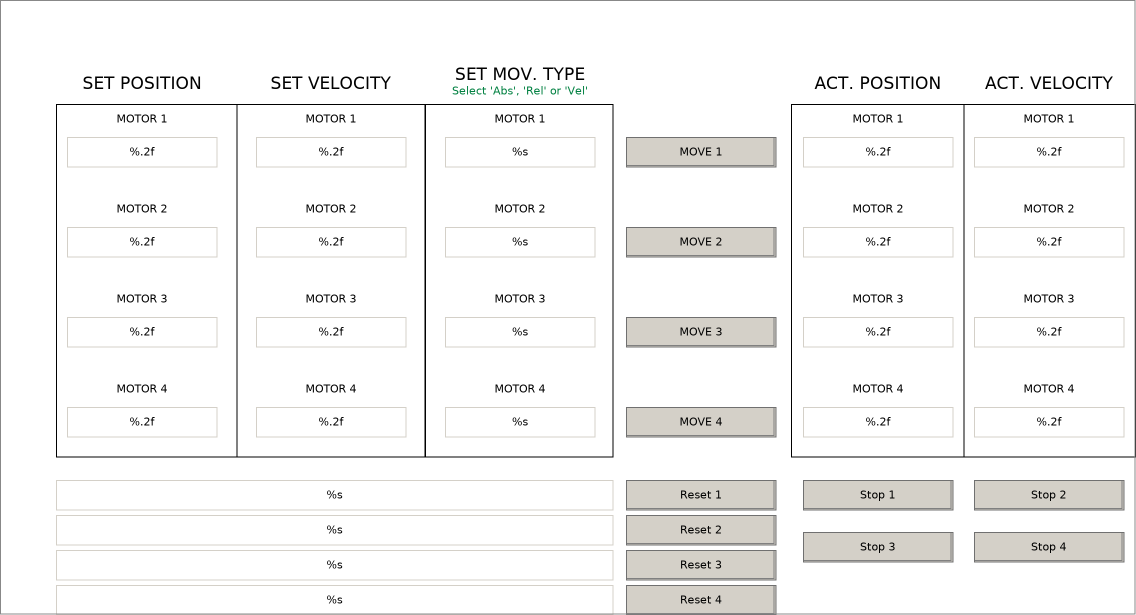
VISUALIZATION Visualization  // 1136x615
    Rectangle (425,104 188x353)
    Rectangle (233,104 192x353)
    Rectangle (56,104 181x353)
    Textfield (67,137 150x30), "%.2f", text variable: MAIN.lrPosition[1]
        OnMouseClick: write the text variable via Default
    Label (67,104 150x30), "MOTOR 1"
    Textfield (67,227 150x30), "%.2f", text variable: MAIN.lrPosition[2]
        OnMouseClick: write the text variable via Default
    Label (67,194 150x30), "MOTOR 2"
    Textfield (67,317 150x30), "%.2f", text variable: MAIN.lrPosition[3]
        OnMouseClick: write the text variable via Default
    Label (67,284 150x30), "MOTOR 3"
    Textfield (67,407 150x30), "%.2f", text variable: MAIN.lrPosition[4]
        OnMouseClick: write the text variable via Default
    Label (67,374 150x30), "MOTOR 4"
    Textfield (256,137 150x30), "%.2f", text variable: MAIN.lrVelocity[1]
        OnMouseClick: write the text variable via Default
    Label (256,104 150x30), "MOTOR 1"
    Textfield (256,227 150x30), "%.2f", text variable: MAIN.lrVelocity[2]
        OnMouseClick: write the text variable via Default
    Label (256,194 150x30), "MOTOR 2"
    Textfield (256,317 150x30), "%.2f", text variable: MAIN.lrVelocity[3]
        OnMouseClick: write the text variable via Default
    Label (256,284 150x30), "MOTOR 3"
    Textfield (256,407 150x30), "%.2f", text variable: MAIN.lrVelocity[4]
        OnMouseClick: write the text variable via Default
    Label (256,374 150x30), "MOTOR 4"
    Textfield (445,137 150x30), "%s", text variable: MAIN.sMovType[1]
        OnMouseClick: write the text variable via Default
    Label (445,104 150x30), "MOTOR 1"
    Textfield (445,227 150x30), "%s", text variable: MAIN.sMovType[2]
        OnMouseClick: write the text variable via Default
    Label (445,194 150x30), "MOTOR 2"
    Textfield (445,317 150x30), "%s", text variable: MAIN.sMovType[3]
        OnMouseClick: write the text variable via Default
    Label (445,284 150x30), "MOTOR 3"
    Textfield (445,407 150x30), "%s", text variable: MAIN.sMovType[4]
        OnMouseClick: write the text variable via Default
    Label (445,374 150x30), "MOTOR 4"
    Label (67,68 150x30), "SET POSITION"
    Label (256,68 150x30), "SET VELOCITY"
    Label (445,59 150x30), "SET MOV. TYPE"
    Rectangle (963,104 173x353)
    Rectangle (791,104 173x353)
    Textfield (803,137 150x30), "%.2f", text variable: MAIN.Motor[1].stat.lrPosActual
    Label (803,104 150x30), "MOTOR 1"
    Textfield (803,227 150x30), "%.2f", text variable: MAIN.Motor[2].stat.lrPosActual
    Label (803,194 150x30), "MOTOR 2"
    Textfield (803,317 150x30), "%.2f", text variable: MAIN.Motor[3].stat.lrPosActual
    Label (803,284 150x30), "MOTOR 3"
    Textfield (803,407 150x30), "%.2f", text variable: MAIN.Motor[4].stat.lrPosActual
    Label (803,374 150x30), "MOTOR 4"
    Textfield (974,137 150x30), "%.2f", text variable: MAIN.Motor[1].stat.lrVelActual
    Label (974,104 150x30), "MOTOR 1"
    Textfield (974,227 150x30), "%.2f", text variable: MAIN.Motor[2].stat.lrVelActual
    Label (974,194 150x30), "MOTOR 2"
    Textfield (974,317 150x30), "%.2f", text variable: MAIN.Motor[3].stat.lrVelActual
    Label (974,284 150x30), "MOTOR 3"
    Textfield (974,407 150x30), "%.2f", text variable: MAIN.Motor[4].stat.lrVelActual
    Label (974,374 150x30), "MOTOR 4"
    Label (803,68 150x30), "ACT. POSITION"
    Label (974,68 150x30), "ACT. VELOCITY"
    Button (626,137 150x30), "MOVE 1"
        tap MAIN.bMove[1] p1329445385=TRUE
    Button (626,227 150x30), "MOVE 2"
        tap MAIN.bMove[2]
    Button (626,317 150x30), "MOVE 3"
        tap MAIN.bMove[3]
    Button (626,407 150x30), "MOVE 4"
        tap MAIN.bMove[4]
    Textfield (56,480 557x30), "%s", text variable: MAIN.sMessage[1]
    Textfield (56,515 557x30), "%s", text variable: MAIN.sMessage[2]
    Textfield (56,550 557x30), "%s", text variable: MAIN.sMessage[3]
    Textfield (56,585 557x30), "%s", text variable: MAIN.sMessage[4]
    Button (626,480 150x30), "Reset 1"
        tap MAIN.bReset[1] p1329445385=TRUE
    Button (626,515 150x30), "Reset 2"
        tap MAIN.bReset[2] p1329445385=TRUE
    Button (626,550 150x30), "Reset 3"
        tap MAIN.bReset[3] p1329445385=TRUE
    Button (626,585 150x30), "Reset 4"
        tap MAIN.bReset[4] p1329445385=TRUE
    Label (445,76 150x30), "Select 'Abs', 'Rel' or 'Vel'"
    Button (803,480 150x30), "Stop 1"
        tap MAIN.bStop[1] p1329445385=TRUE
    Button (974,480 150x30), "Stop 2"
        tap MAIN.bStop[2] p1329445385=TRUE
    Button (803,532 150x30), "Stop 3"
        tap MAIN.bStop[3] p1329445385=TRUE
    Button (974,532 150x30), "Stop 4"
        tap MAIN.bStop[4] p1329445385=TRUE
END_VISUALIZATION

(* stored: Version 1.1.0.1, ProductVersion 3.1.4024.9
   Visu Visualization: Id {2949dbbf-af8e-4a5d-be44-249490d97200} *)
